{attribute addProperty BoxType "EL4002-0000-0018"}
{attribute addProperty Id "AO_Output_ChannelAT %Q*ARRAY[0..1] OF AO_Output_Channel_F57FA4F93240WcStateAT %I*WcState_64F6A8C6810InfoDataAT %I*InfoData_BC63D37F80100"}
{attribute addProperty CRC "1402100183"}
{attribute addProperty SizeInBites "120"}
{attribute addProperty SizeInBytes "15"}
TYPE EL4002_F05A29F1 :
STRUCT
	{attribute addProperty Name "AO_Output_Channel"}
	AO_Output_Channel : ARRAY[0..1] OF AO_Output_Channel_F57FA4F9;
	{attribute addProperty Name "WcState"}
	WcState : WcState_64F6A8C6;
	{attribute addProperty Name "InfoData"}
	InfoData : InfoData_BC63D37F;
END_STRUCT
END_TYPE

(* stored: Version 1.2.0.0, ProductVersion 3.1.4024.9
   DUT EL4002_F05A29F1: Id {87d20b0d-2b68-4a8b-a854-9f30d8f3aa68} *)
